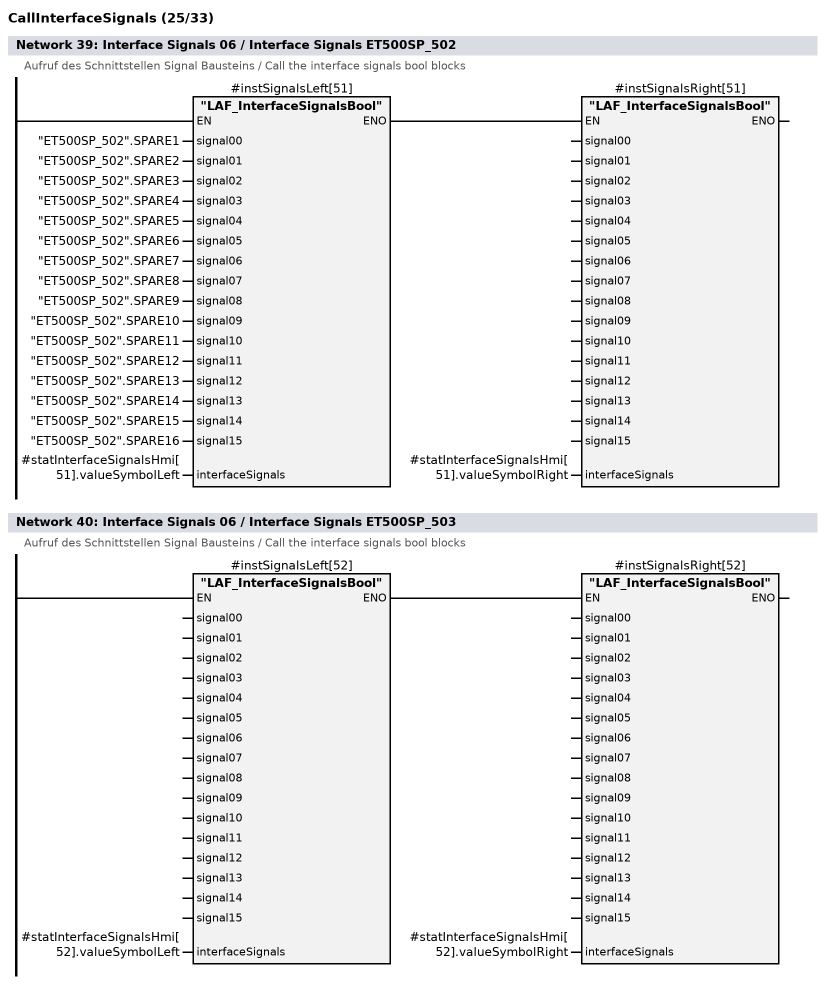
   RUNG wire#powerrail
      #instSignalsLeft[51](signal00 := "ET500SP_502".SPARE1, signal01 := "ET500SP_502".SPARE2, signal02 := "ET500SP_502".SPARE3, signal03 := "ET500SP_502".SPARE4, signal04 := "ET500SP_502".SPARE5, signal05 := "ET500SP_502".SPARE6, signal06 := "ET500SP_502".SPARE7, signal07 := "ET500SP_502".SPARE8, signal08 := "ET500SP_502".SPARE9, signal09 := "ET500SP_502".SPARE10, signal10 := "ET500SP_502".SPARE11, signal11 := "ET500SP_502".SPARE12, signal12 := "ET500SP_502".SPARE13, signal13 := "ET500SP_502".SPARE14, signal14 := "ET500SP_502".SPARE15, signal15 := "ET500SP_502".SPARE16, interfaceSignals := #statInterfaceSignalsHmi[51].valueSymbolLeft)
      #instSignalsRight[51](signal00 :=, signal01 :=, signal02 :=, signal03 :=, signal04 :=, signal05 :=, signal06 :=, signal07 :=, signal08 :=, signal09 :=, signal10 :=, signal11 :=, signal12 :=, signal13 :=, signal14 :=, signal15 :=, interfaceSignals := #statInterfaceSignalsHmi[51].valueSymbolRight)
   END_RUNG
   // the same network as SCL:
   #instSignalsLeft[51](signal00 := "ET500SP_502".SPARE1,   // "LAF_InterfaceSignalsBool"
                        signal01 := "ET500SP_502".SPARE2,
                        signal02 := "ET500SP_502".SPARE3,
                        signal03 := "ET500SP_502".SPARE4,
                        signal04 := "ET500SP_502".SPARE5,
                        signal05 := "ET500SP_502".SPARE6,
                        signal06 := "ET500SP_502".SPARE7,
                        signal07 := "ET500SP_502".SPARE8,
                        signal08 := "ET500SP_502".SPARE9,
                        signal09 := "ET500SP_502".SPARE10,
                        signal10 := "ET500SP_502".SPARE11,
                        signal11 := "ET500SP_502".SPARE12,
                        signal12 := "ET500SP_502".SPARE13,
                        signal13 := "ET500SP_502".SPARE14,
                        signal14 := "ET500SP_502".SPARE15,
                        signal15 := "ET500SP_502".SPARE16,
                        interfaceSignals := #statInterfaceSignalsHmi[51].valueSymbolLeft,
                        ENO => #_w1);
   IF #_w1 THEN
       #instSignalsRight[51](interfaceSignals := #statInterfaceSignalsHmi[51].valueSymbolRight);   // "LAF_InterfaceSignalsBool"
   END_IF;
END_REGION

REGION Network 40: Interface Signals 06 / Interface Signals ET500SP_503
   // Aufruf des Schnittstellen Signal Bausteins / Call the interface signals bool blocks
   RUNG wire#powerrail
      #instSignalsLeft[52](signal00 :=, signal01 :=, signal02 :=, signal03 :=, signal04 :=, signal05 :=, signal06 :=, signal07 :=, signal08 :=, signal09 :=, signal10 :=, signal11 :=, signal12 :=, signal13 :=, signal14 :=, signal15 :=, interfaceSignals := #statInterfaceSignalsHmi[52].valueSymbolLeft)
      #instSignalsRight[52](signal00 :=, signal01 :=, signal02 :=, signal03 :=, signal04 :=, signal05 :=, signal06 :=, signal07 :=, signal08 :=, signal09 :=, signal10 :=, signal11 :=, signal12 :=, signal13 :=, signal14 :=, signal15 :=, interfaceSignals := #statInterfaceSignalsHmi[52].valueSymbolRight)
   END_RUNG
   // the same network as SCL:
   #instSignalsLeft[52](interfaceSignals := #statInterfaceSignalsHmi[52].valueSymbolLeft, ENO => #_w1);   // "LAF_InterfaceSignalsBool"
   IF #_w1 THEN
       #instSignalsRight[52](interfaceSignals := #statInterfaceSignalsHmi[52].valueSymbolRight);   // "LAF_InterfaceSignalsBool"
   END_IF;
END_REGION

REGION Network 41: Interface Signals 06 / Interface Signals ET500SP_504
   // Aufruf des Schnittstellen Signal Bausteins / Call the interface signals bool blocks
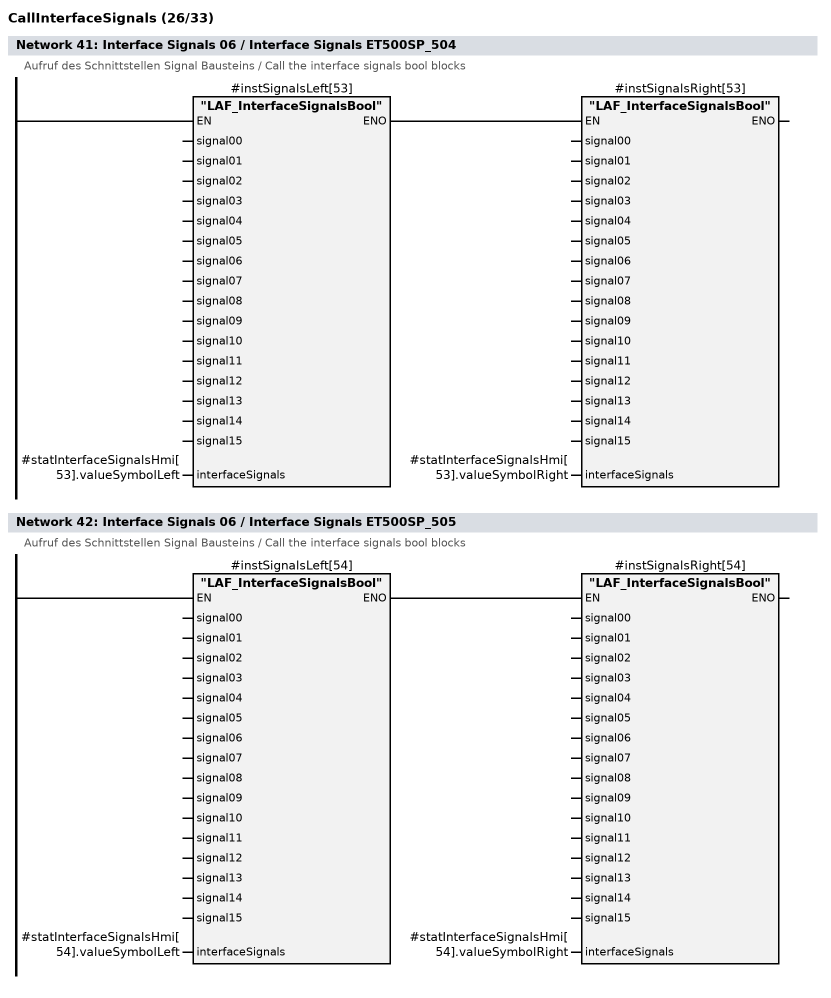
   RUNG wire#powerrail
      #instSignalsLeft[53](signal00 :=, signal01 :=, signal02 :=, signal03 :=, signal04 :=, signal05 :=, signal06 :=, signal07 :=, signal08 :=, signal09 :=, signal10 :=, signal11 :=, signal12 :=, signal13 :=, signal14 :=, signal15 :=, interfaceSignals := #statInterfaceSignalsHmi[53].valueSymbolLeft)
      #instSignalsRight[53](signal00 :=, signal01 :=, signal02 :=, signal03 :=, signal04 :=, signal05 :=, signal06 :=, signal07 :=, signal08 :=, signal09 :=, signal10 :=, signal11 :=, signal12 :=, signal13 :=, signal14 :=, signal15 :=, interfaceSignals := #statInterfaceSignalsHmi[53].valueSymbolRight)
   END_RUNG
   // the same network as SCL:
   #instSignalsLeft[53](interfaceSignals := #statInterfaceSignalsHmi[53].valueSymbolLeft, ENO => #_w1);   // "LAF_InterfaceSignalsBool"
   IF #_w1 THEN
       #instSignalsRight[53](interfaceSignals := #statInterfaceSignalsHmi[53].valueSymbolRight);   // "LAF_InterfaceSignalsBool"
   END_IF;
END_REGION

REGION Network 42: Interface Signals 06 / Interface Signals ET500SP_505
   // Aufruf des Schnittstellen Signal Bausteins / Call the interface signals bool blocks
   RUNG wire#powerrail
      #instSignalsLeft[54](signal00 :=, signal01 :=, signal02 :=, signal03 :=, signal04 :=, signal05 :=, signal06 :=, signal07 :=, signal08 :=, signal09 :=, signal10 :=, signal11 :=, signal12 :=, signal13 :=, signal14 :=, signal15 :=, interfaceSignals := #statInterfaceSignalsHmi[54].valueSymbolLeft)
      #instSignalsRight[54](signal00 :=, signal01 :=, signal02 :=, signal03 :=, signal04 :=, signal05 :=, signal06 :=, signal07 :=, signal08 :=, signal09 :=, signal10 :=, signal11 :=, signal12 :=, signal13 :=, signal14 :=, signal15 :=, interfaceSignals := #statInterfaceSignalsHmi[54].valueSymbolRight)
   END_RUNG
   // the same network as SCL:
   #instSignalsLeft[54](interfaceSignals := #statInterfaceSignalsHmi[54].valueSymbolLeft, ENO => #_w1);   // "LAF_InterfaceSignalsBool"
   IF #_w1 THEN
       #instSignalsRight[54](interfaceSignals := #statInterfaceSignalsHmi[54].valueSymbolRight);   // "LAF_InterfaceSignalsBool"
   END_IF;
END_REGION

REGION Network 43: Interface Signals 06 / Interface Signals ET500SP_506
   // Aufruf des Schnittstellen Signal Bausteins / Call the interface signals bool blocks
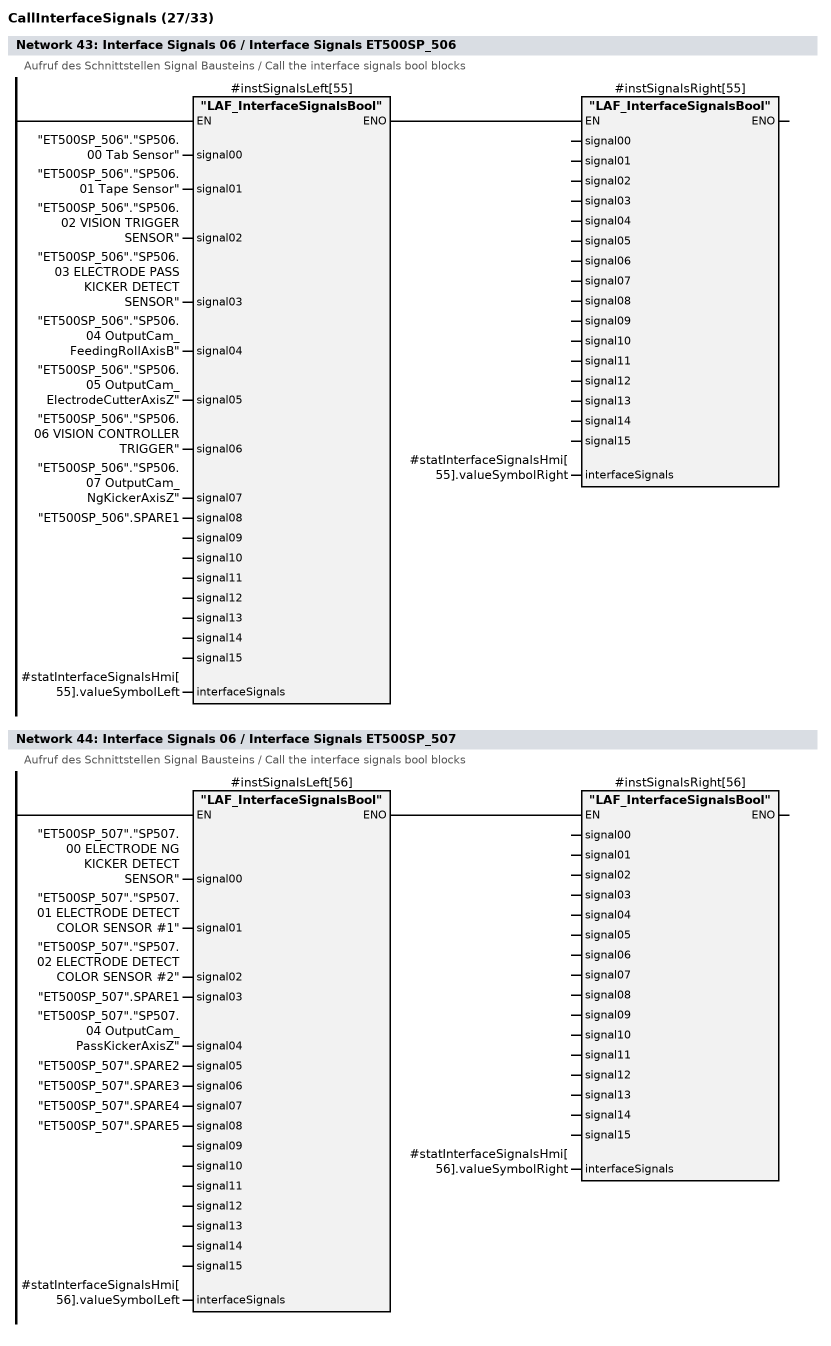
   RUNG wire#powerrail
      #instSignalsLeft[55](signal00 := "ET500SP_506"."SP506.00 Tab Sensor", signal01 := "ET500SP_506"."SP506.01 Tape Sensor", signal02 := "ET500SP_506"."SP506.02 VISION TRIGGER SENSOR", signal03 := "ET500SP_506"."SP506.03 ELECTRODE PASS KICKER DETECT SENSOR", signal04 := "ET500SP_506"."SP506.04 OutputCam_FeedingRollAxisB", signal05 := "ET500SP_506"."SP506.05 OutputCam_ElectrodeCutterAxisZ", signal06 := "ET500SP_506"."SP506.06 VISION CONTROLLER TRIGGER", signal07 := "ET500SP_506"."SP506.07 OutputCam_NgKickerAxisZ", signal08 := "ET500SP_506".SPARE1, signal09 :=, signal10 :=, signal11 :=, signal12 :=, signal13 :=, signal14 :=, signal15 :=, interfaceSignals := #statInterfaceSignalsHmi[55].valueSymbolLeft)
      #instSignalsRight[55](signal00 :=, signal01 :=, signal02 :=, signal03 :=, signal04 :=, signal05 :=, signal06 :=, signal07 :=, signal08 :=, signal09 :=, signal10 :=, signal11 :=, signal12 :=, signal13 :=, signal14 :=, signal15 :=, interfaceSignals := #statInterfaceSignalsHmi[55].valueSymbolRight)
   END_RUNG
   // the same network as SCL:
   #instSignalsLeft[55](signal00 := "ET500SP_506"."SP506.00 Tab Sensor",   // "LAF_InterfaceSignalsBool"
                        signal01 := "ET500SP_506"."SP506.01 Tape Sensor",
                        signal02 := "ET500SP_506"."SP506.02 VISION TRIGGER SENSOR",
                        signal03 := "ET500SP_506"."SP506.03 ELECTRODE PASS KICKER DETECT SENSOR",
                        signal04 := "ET500SP_506"."SP506.04 OutputCam_FeedingRollAxisB",
                        signal05 := "ET500SP_506"."SP506.05 OutputCam_ElectrodeCutterAxisZ",
                        signal06 := "ET500SP_506"."SP506.06 VISION CONTROLLER TRIGGER",
                        signal07 := "ET500SP_506"."SP506.07 OutputCam_NgKickerAxisZ",
                        signal08 := "ET500SP_506".SPARE1,
                        interfaceSignals := #statInterfaceSignalsHmi[55].valueSymbolLeft,
                        ENO => #_w1);
   IF #_w1 THEN
       #instSignalsRight[55](interfaceSignals := #statInterfaceSignalsHmi[55].valueSymbolRight);   // "LAF_InterfaceSignalsBool"
   END_IF;
END_REGION

REGION Network 44: Interface Signals 06 / Interface Signals ET500SP_507
   // Aufruf des Schnittstellen Signal Bausteins / Call the interface signals bool blocks
   RUNG wire#powerrail
      #instSignalsLeft[56](signal00 := "ET500SP_507"."SP507.00 ELECTRODE NG KICKER DETECT SENSOR", signal01 := "ET500SP_507"."SP507.01 ELECTRODE DETECT COLOR SENSOR #1", signal02 := "ET500SP_507"."SP507.02 ELECTRODE DETECT COLOR SENSOR #2", signal03 := "ET500SP_507".SPARE1, signal04 := "ET500SP_507"."SP507.04 OutputCam_PassKickerAxisZ", signal05 := "ET500SP_507".SPARE2, signal06 := "ET500SP_507".SPARE3, signal07 := "ET500SP_507".SPARE4, signal08 := "ET500SP_507".SPARE5, signal09 :=, signal10 :=, signal11 :=, signal12 :=, signal13 :=, signal14 :=, signal15 :=, interfaceSignals := #statInterfaceSignalsHmi[56].valueSymbolLeft)
      #instSignalsRight[56](signal00 :=, signal01 :=, signal02 :=, signal03 :=, signal04 :=, signal05 :=, signal06 :=, signal07 :=, signal08 :=, signal09 :=, signal10 :=, signal11 :=, signal12 :=, signal13 :=, signal14 :=, signal15 :=, interfaceSignals := #statInterfaceSignalsHmi[56].valueSymbolRight)
   END_RUNG
   // the same network as SCL:
   #instSignalsLeft[56](signal00 := "ET500SP_507"."SP507.00 ELECTRODE NG KICKER DETECT SENSOR",   // "LAF_InterfaceSignalsBool"
                        signal01 := "ET500SP_507"."SP507.01 ELECTRODE DETECT COLOR SENSOR #1",
                        signal02 := "ET500SP_507"."SP507.02 ELECTRODE DETECT COLOR SENSOR #2",
                        signal03 := "ET500SP_507".SPARE1,
                        signal04 := "ET500SP_507"."SP507.04 OutputCam_PassKickerAxisZ",
                        signal05 := "ET500SP_507".SPARE2,
                        signal06 := "ET500SP_507".SPARE3,
                        signal07 := "ET500SP_507".SPARE4,
                        signal08 := "ET500SP_507".SPARE5,
                        interfaceSignals := #statInterfaceSignalsHmi[56].valueSymbolLeft,
                        ENO => #_w1);
   IF #_w1 THEN
       #instSignalsRight[56](interfaceSignals := #statInterfaceSignalsHmi[56].valueSymbolRight);   // "LAF_InterfaceSignalsBool"
   END_IF;
END_REGION

REGION Network 45: Interface Signals 06 / Interface Signals ET500SP_508
   // Aufruf des Schnittstellen Signal Bausteins / Call the interface signals bool blocks
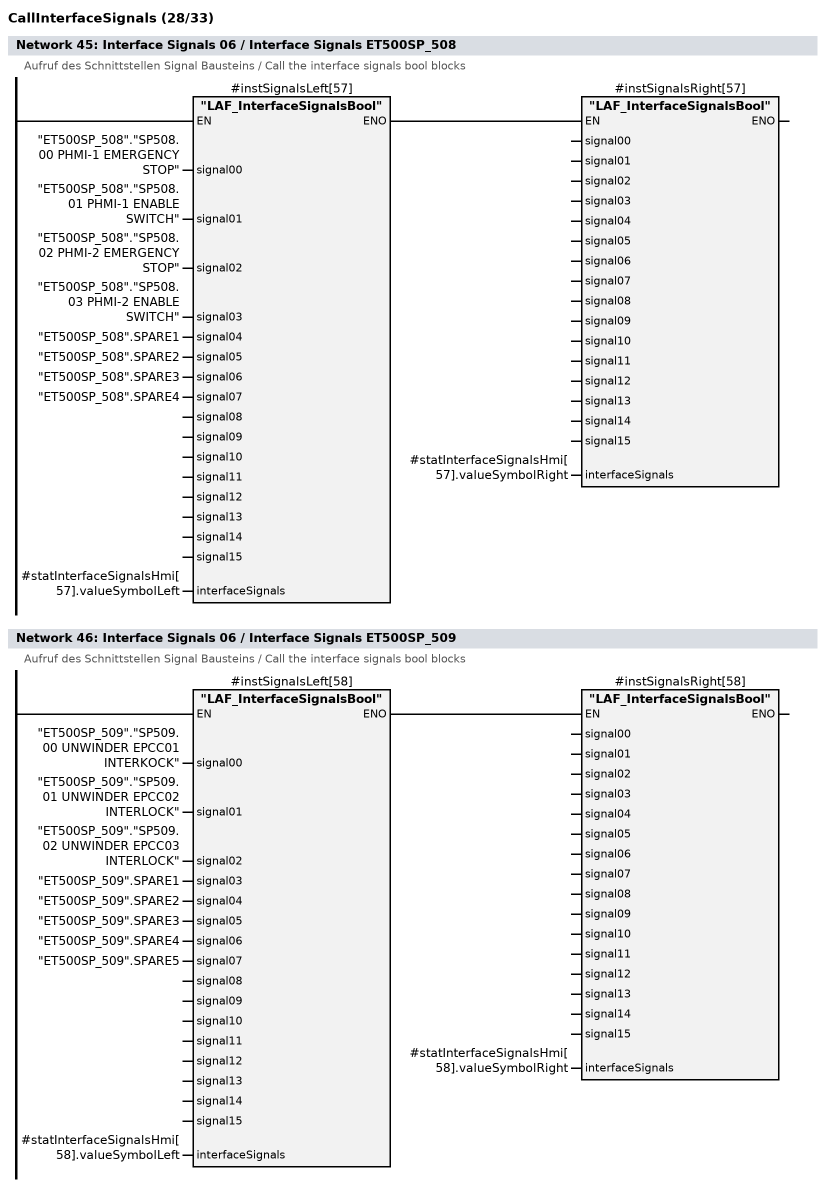
   RUNG wire#powerrail
      #instSignalsLeft[57](signal00 := "ET500SP_508"."SP508.00 PHMI-1 EMERGENCY STOP", signal01 := "ET500SP_508"."SP508.01 PHMI-1 ENABLE SWITCH", signal02 := "ET500SP_508"."SP508.02 PHMI-2 EMERGENCY STOP", signal03 := "ET500SP_508"."SP508.03 PHMI-2 ENABLE SWITCH", signal04 := "ET500SP_508".SPARE1, signal05 := "ET500SP_508".SPARE2, signal06 := "ET500SP_508".SPARE3, signal07 := "ET500SP_508".SPARE4, signal08 :=, signal09 :=, signal10 :=, signal11 :=, signal12 :=, signal13 :=, signal14 :=, signal15 :=, interfaceSignals := #statInterfaceSignalsHmi[57].valueSymbolLeft)
      #instSignalsRight[57](signal00 :=, signal01 :=, signal02 :=, signal03 :=, signal04 :=, signal05 :=, signal06 :=, signal07 :=, signal08 :=, signal09 :=, signal10 :=, signal11 :=, signal12 :=, signal13 :=, signal14 :=, signal15 :=, interfaceSignals := #statInterfaceSignalsHmi[57].valueSymbolRight)
   END_RUNG
   // the same network as SCL:
   #instSignalsLeft[57](signal00 := "ET500SP_508"."SP508.00 PHMI-1 EMERGENCY STOP",   // "LAF_InterfaceSignalsBool"
                        signal01 := "ET500SP_508"."SP508.01 PHMI-1 ENABLE SWITCH",
                        signal02 := "ET500SP_508"."SP508.02 PHMI-2 EMERGENCY STOP",
                        signal03 := "ET500SP_508"."SP508.03 PHMI-2 ENABLE SWITCH",
                        signal04 := "ET500SP_508".SPARE1,
                        signal05 := "ET500SP_508".SPARE2,
                        signal06 := "ET500SP_508".SPARE3,
                        signal07 := "ET500SP_508".SPARE4,
                        interfaceSignals := #statInterfaceSignalsHmi[57].valueSymbolLeft,
                        ENO => #_w1);
   IF #_w1 THEN
       #instSignalsRight[57](interfaceSignals := #statInterfaceSignalsHmi[57].valueSymbolRight);   // "LAF_InterfaceSignalsBool"
   END_IF;
END_REGION

REGION Network 46: Interface Signals 06 / Interface Signals ET500SP_509
   // Aufruf des Schnittstellen Signal Bausteins / Call the interface signals bool blocks
   RUNG wire#powerrail
      #instSignalsLeft[58](signal00 := "ET500SP_509"."SP509.00 UNWINDER EPCC01 INTERKOCK", signal01 := "ET500SP_509"."SP509.01 UNWINDER EPCC02 INTERLOCK", signal02 := "ET500SP_509"."SP509.02 UNWINDER EPCC03 INTERLOCK", signal03 := "ET500SP_509".SPARE1, signal04 := "ET500SP_509".SPARE2, signal05 := "ET500SP_509".SPARE3, signal06 := "ET500SP_509".SPARE4, signal07 := "ET500SP_509".SPARE5, signal08 :=, signal09 :=, signal10 :=, signal11 :=, signal12 :=, signal13 :=, signal14 :=, signal15 :=, interfaceSignals := #statInterfaceSignalsHmi[58].valueSymbolLeft)
      #instSignalsRight[58](signal00 :=, signal01 :=, signal02 :=, signal03 :=, signal04 :=, signal05 :=, signal06 :=, signal07 :=, signal08 :=, signal09 :=, signal10 :=, signal11 :=, signal12 :=, signal13 :=, signal14 :=, signal15 :=, interfaceSignals := #statInterfaceSignalsHmi[58].valueSymbolRight)
   END_RUNG
   // the same network as SCL:
   #instSignalsLeft[58](signal00 := "ET500SP_509"."SP509.00 UNWINDER EPCC01 INTERKOCK",   // "LAF_InterfaceSignalsBool"
                        signal01 := "ET500SP_509"."SP509.01 UNWINDER EPCC02 INTERLOCK",
                        signal02 := "ET500SP_509"."SP509.02 UNWINDER EPCC03 INTERLOCK",
                        signal03 := "ET500SP_509".SPARE1,
                        signal04 := "ET500SP_509".SPARE2,
                        signal05 := "ET500SP_509".SPARE3,
                        signal06 := "ET500SP_509".SPARE4,
                        signal07 := "ET500SP_509".SPARE5,
                        interfaceSignals := #statInterfaceSignalsHmi[58].valueSymbolLeft,
                        ENO => #_w1);
   IF #_w1 THEN
       #instSignalsRight[58](interfaceSignals := #statInterfaceSignalsHmi[58].valueSymbolRight);   // "LAF_InterfaceSignalsBool"
   END_IF;
END_REGION

REGION Network 47: Interface Signals 06 / Interface Signals ET500SP_513
   // Aufruf des Schnittstellen Signal Bausteins / Call the interface signals bool blocks
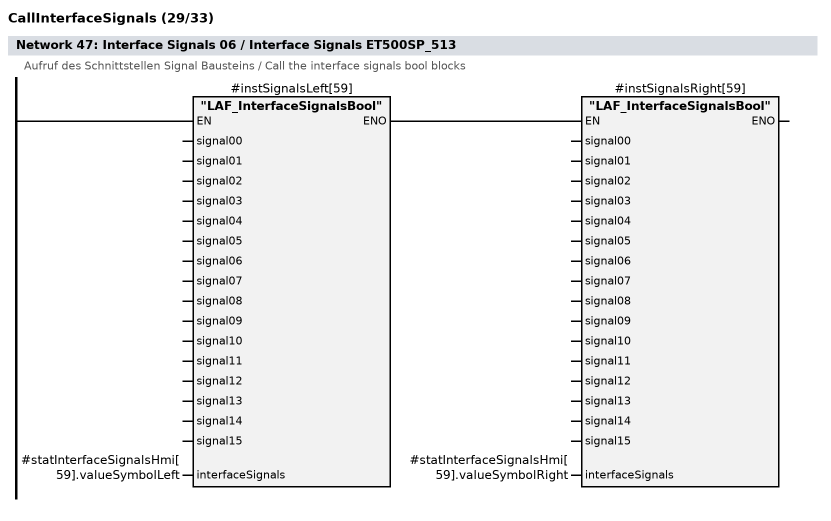
   RUNG wire#powerrail
      #instSignalsLeft[59](signal00 :=, signal01 :=, signal02 :=, signal03 :=, signal04 :=, signal05 :=, signal06 :=, signal07 :=, signal08 :=, signal09 :=, signal10 :=, signal11 :=, signal12 :=, signal13 :=, signal14 :=, signal15 :=, interfaceSignals := #statInterfaceSignalsHmi[59].valueSymbolLeft)
      #instSignalsRight[59](signal00 :=, signal01 :=, signal02 :=, signal03 :=, signal04 :=, signal05 :=, signal06 :=, signal07 :=, signal08 :=, signal09 :=, signal10 :=, signal11 :=, signal12 :=, signal13 :=, signal14 :=, signal15 :=, interfaceSignals := #statInterfaceSignalsHmi[59].valueSymbolRight)
   END_RUNG
   // the same network as SCL:
   #instSignalsLeft[59](interfaceSignals := #statInterfaceSignalsHmi[59].valueSymbolLeft, ENO => #_w1);   // "LAF_InterfaceSignalsBool"
   IF #_w1 THEN
       #instSignalsRight[59](interfaceSignals := #statInterfaceSignalsHmi[59].valueSymbolRight);   // "LAF_InterfaceSignalsBool"
   END_IF;
END_REGION

REGION Network 48: Interface Signals 06 / Interface Signals CPU DI1
   // Aufruf des Schnittstellen Signal Bausteins / Call the interface signals bool blocks
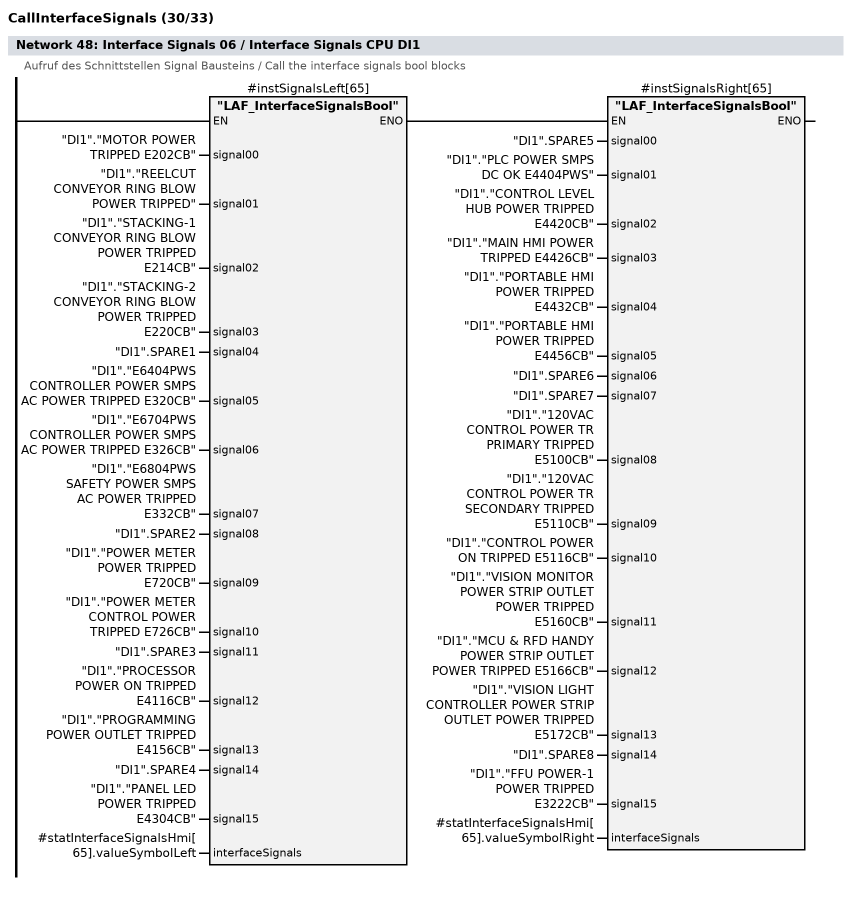
   RUNG wire#powerrail
      #instSignalsLeft[65](signal00 := "DI1"."MOTOR POWER TRIPPED E202CB", signal01 := "DI1"."REELCUT CONVEYOR RING BLOW POWER TRIPPED", signal02 := "DI1"."STACKING-1 CONVEYOR RING BLOW POWER TRIPPED E214CB", signal03 := "DI1"."STACKING-2 CONVEYOR RING BLOW POWER TRIPPED E220CB", signal04 := "DI1".SPARE1, signal05 := "DI1"."E6404PWS CONTROLLER POWER SMPS AC POWER TRIPPED E320CB", signal06 := "DI1"."E6704PWS CONTROLLER POWER SMPS AC POWER TRIPPED E326CB", signal07 := "DI1"."E6804PWS SAFETY POWER SMPS AC POWER TRIPPED E332CB", signal08 := "DI1".SPARE2, signal09 := "DI1"."POWER METER POWER TRIPPED E720CB", signal10 := "DI1"."POWER METER CONTROL POWER TRIPPED E726CB", signal11 := "DI1".SPARE3, signal12 := "DI1"."PROCESSOR POWER ON TRIPPED E4116CB", signal13 := "DI1"."PROGRAMMING POWER OUTLET TRIPPED E4156CB", signal14 := "DI1".SPARE4, signal15 := "DI1"."PANEL LED POWER TRIPPED E4304CB", interfaceSignals := #statInterfaceSignalsHmi[65].valueSymbolLeft)
      #instSignalsRight[65](signal00 := "DI1".SPARE5, signal01 := "DI1"."PLC POWER SMPS DC OK E4404PWS", signal02 := "DI1"."CONTROL LEVEL HUB POWER TRIPPED E4420CB", signal03 := "DI1"."MAIN HMI POWER TRIPPED E4426CB", signal04 := "DI1"."PORTABLE HMI POWER TRIPPED E4432CB", signal05 := "DI1"."PORTABLE HMI POWER TRIPPED E4456CB", signal06 := "DI1".SPARE6, signal07 := "DI1".SPARE7, signal08 := "DI1"."120VAC CONTROL POWER TR PRIMARY TRIPPED E5100CB", signal09 := "DI1"."120VAC CONTROL POWER TR SECONDARY TRIPPED E5110CB", signal10 := "DI1"."CONTROL POWER ON TRIPPED E5116CB", signal11 := "DI1"."VISION MONITOR POWER STRIP OUTLET POWER TRIPPED E5160CB", signal12 := "DI1"."MCU & RFD HANDY POWER STRIP OUTLET POWER TRIPPED E5166CB", signal13 := "DI1"."VISION LIGHT CONTROLLER POWER STRIP OUTLET POWER TRIPPED E5172CB", signal14 := "DI1".SPARE8, signal15 := "DI1"."FFU POWER-1 POWER TRIPPED E3222CB", interfaceSignals := #statInterfaceSignalsHmi[65].valueSymbolRight)
   END_RUNG
   // the same network as SCL:
   #instSignalsLeft[65](signal00 := "DI1"."MOTOR POWER TRIPPED E202CB",   // "LAF_InterfaceSignalsBool"
                        signal01 := "DI1"."REELCUT CONVEYOR RING BLOW POWER TRIPPED",
                        signal02 := "DI1"."STACKING-1 CONVEYOR RING BLOW POWER TRIPPED E214CB",
                        signal03 := "DI1"."STACKING-2 CONVEYOR RING BLOW POWER TRIPPED E220CB",
                        signal04 := "DI1".SPARE1,
                        signal05 := "DI1"."E6404PWS CONTROLLER POWER SMPS AC POWER TRIPPED E320CB",
                        signal06 := "DI1"."E6704PWS CONTROLLER POWER SMPS AC POWER TRIPPED E326CB",
                        signal07 := "DI1"."E6804PWS SAFETY POWER SMPS AC POWER TRIPPED E332CB",
                        signal08 := "DI1".SPARE2,
                        signal09 := "DI1"."POWER METER POWER TRIPPED E720CB",
                        signal10 := "DI1"."POWER METER CONTROL POWER TRIPPED E726CB",
                        signal11 := "DI1".SPARE3,
                        signal12 := "DI1"."PROCESSOR POWER ON TRIPPED E4116CB",
                        signal13 := "DI1"."PROGRAMMING POWER OUTLET TRIPPED E4156CB",
                        signal14 := "DI1".SPARE4,
                        signal15 := "DI1"."PANEL LED POWER TRIPPED E4304CB",
                        interfaceSignals := #statInterfaceSignalsHmi[65].valueSymbolLeft,
                        ENO => #_w1);
   IF #_w1 THEN
       #instSignalsRight[65](signal00 := "DI1".SPARE5,   // "LAF_InterfaceSignalsBool"
                             signal01 := "DI1"."PLC POWER SMPS DC OK E4404PWS",
                             signal02 := "DI1"."CONTROL LEVEL HUB POWER TRIPPED E4420CB",
                             signal03 := "DI1"."MAIN HMI POWER TRIPPED E4426CB",
                             signal04 := "DI1"."PORTABLE HMI POWER TRIPPED E4432CB",
                             signal05 := "DI1"."PORTABLE HMI POWER TRIPPED E4456CB",
                             signal06 := "DI1".SPARE6,
                             signal07 := "DI1".SPARE7,
                             signal08 := "DI1"."120VAC CONTROL POWER TR PRIMARY TRIPPED E5100CB",
                             signal09 := "DI1"."120VAC CONTROL POWER TR SECONDARY TRIPPED E5110CB",
                             signal10 := "DI1"."CONTROL POWER ON TRIPPED E5116CB",
                             signal11 := "DI1"."VISION MONITOR POWER STRIP OUTLET POWER TRIPPED E5160CB",
                             signal12 := "DI1"."MCU & RFD HANDY POWER STRIP OUTLET POWER TRIPPED E5166CB",
                             signal13 := "DI1"."VISION LIGHT CONTROLLER POWER STRIP OUTLET POWER TRIPPED E5172CB",
                             signal14 := "DI1".SPARE8,
                             signal15 := "DI1"."FFU POWER-1 POWER TRIPPED E3222CB",
                             interfaceSignals := #statInterfaceSignalsHmi[65].valueSymbolRight);
   END_IF;
END_REGION

REGION Network 49: Interface Signals 06 / Interface Signals CPU DI2
   // Aufruf des Schnittstellen Signal Bausteins / Call the interface signals bool blocks
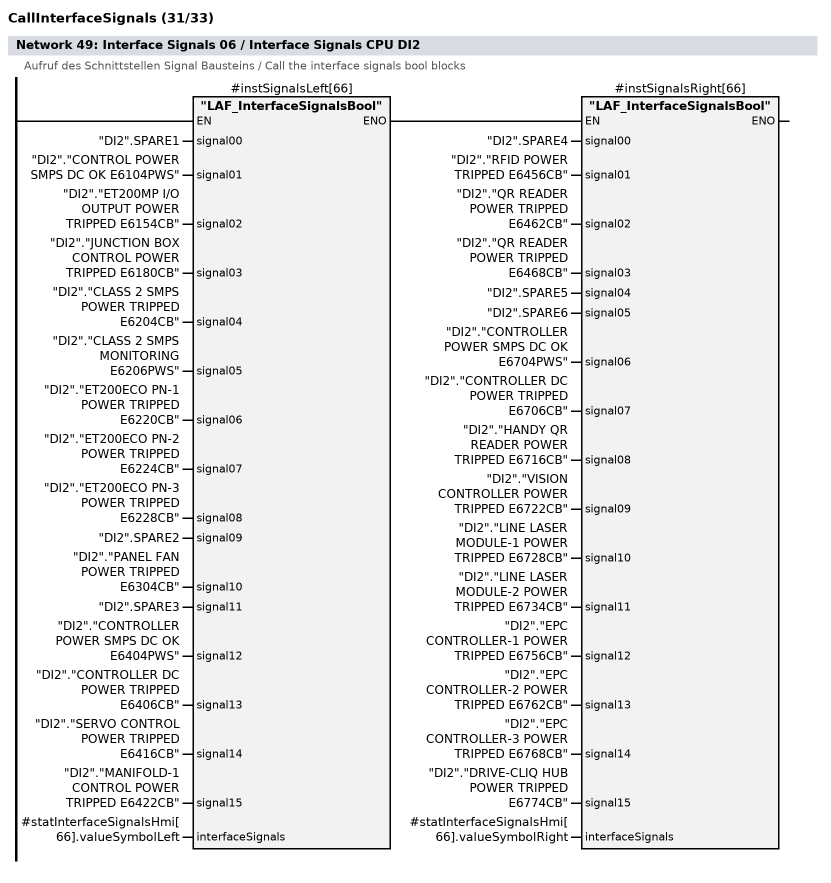
   RUNG wire#powerrail
      #instSignalsLeft[66](signal00 := "DI2".SPARE1, signal01 := "DI2"."CONTROL POWER SMPS DC OK E6104PWS", signal02 := "DI2"."ET200MP I/O OUTPUT POWER TRIPPED E6154CB", signal03 := "DI2"."JUNCTION BOX CONTROL POWER TRIPPED E6180CB", signal04 := "DI2"."CLASS 2 SMPS POWER TRIPPED E6204CB", signal05 := "DI2"."CLASS 2 SMPS MONITORING E6206PWS", signal06 := "DI2"."ET200ECO PN-1 POWER TRIPPED E6220CB", signal07 := "DI2"."ET200ECO PN-2 POWER TRIPPED E6224CB", signal08 := "DI2"."ET200ECO PN-3 POWER TRIPPED E6228CB", signal09 := "DI2".SPARE2, signal10 := "DI2"."PANEL FAN POWER TRIPPED E6304CB", signal11 := "DI2".SPARE3, signal12 := "DI2"."CONTROLLER POWER SMPS DC OK E6404PWS", signal13 := "DI2"."CONTROLLER DC POWER TRIPPED E6406CB", signal14 := "DI2"."SERVO CONTROL POWER TRIPPED E6416CB", signal15 := "DI2"."MANIFOLD-1 CONTROL POWER TRIPPED E6422CB", interfaceSignals := #statInterfaceSignalsHmi[66].valueSymbolLeft)
      #instSignalsRight[66](signal00 := "DI2".SPARE4, signal01 := "DI2"."RFID POWER TRIPPED E6456CB", signal02 := "DI2"."QR READER POWER TRIPPED E6462CB", signal03 := "DI2"."QR READER POWER TRIPPED E6468CB", signal04 := "DI2".SPARE5, signal05 := "DI2".SPARE6, signal06 := "DI2"."CONTROLLER POWER SMPS DC OK E6704PWS", signal07 := "DI2"."CONTROLLER DC POWER TRIPPED E6706CB", signal08 := "DI2"."HANDY QR READER POWER TRIPPED E6716CB", signal09 := "DI2"."VISION CONTROLLER POWER TRIPPED E6722CB", signal10 := "DI2"."LINE LASER MODULE-1 POWER TRIPPED E6728CB", signal11 := "DI2"."LINE LASER MODULE-2 POWER TRIPPED E6734CB", signal12 := "DI2"."EPC CONTROLLER-1 POWER TRIPPED E6756CB", signal13 := "DI2"."EPC CONTROLLER-2 POWER TRIPPED E6762CB", signal14 := "DI2"."EPC CONTROLLER-3 POWER TRIPPED E6768CB", signal15 := "DI2"."DRIVE-CLIQ HUB POWER TRIPPED E6774CB", interfaceSignals := #statInterfaceSignalsHmi[66].valueSymbolRight)
   END_RUNG
   // the same network as SCL:
   #instSignalsLeft[66](signal00 := "DI2".SPARE1,   // "LAF_InterfaceSignalsBool"
                        signal01 := "DI2"."CONTROL POWER SMPS DC OK E6104PWS",
                        signal02 := "DI2"."ET200MP I/O OUTPUT POWER TRIPPED E6154CB",
                        signal03 := "DI2"."JUNCTION BOX CONTROL POWER TRIPPED E6180CB",
                        signal04 := "DI2"."CLASS 2 SMPS POWER TRIPPED E6204CB",
                        signal05 := "DI2"."CLASS 2 SMPS MONITORING E6206PWS",
                        signal06 := "DI2"."ET200ECO PN-1 POWER TRIPPED E6220CB",
                        signal07 := "DI2"."ET200ECO PN-2 POWER TRIPPED E6224CB",
                        signal08 := "DI2"."ET200ECO PN-3 POWER TRIPPED E6228CB",
                        signal09 := "DI2".SPARE2,
                        signal10 := "DI2"."PANEL FAN POWER TRIPPED E6304CB",
                        signal11 := "DI2".SPARE3,
                        signal12 := "DI2"."CONTROLLER POWER SMPS DC OK E6404PWS",
                        signal13 := "DI2"."CONTROLLER DC POWER TRIPPED E6406CB",
                        signal14 := "DI2"."SERVO CONTROL POWER TRIPPED E6416CB",
                        signal15 := "DI2"."MANIFOLD-1 CONTROL POWER TRIPPED E6422CB",
                        interfaceSignals := #statInterfaceSignalsHmi[66].valueSymbolLeft,
                        ENO => #_w1);
   IF #_w1 THEN
       #instSignalsRight[66](signal00 := "DI2".SPARE4,   // "LAF_InterfaceSignalsBool"
                             signal01 := "DI2"."RFID POWER TRIPPED E6456CB",
                             signal02 := "DI2"."QR READER POWER TRIPPED E6462CB",
                             signal03 := "DI2"."QR READER POWER TRIPPED E6468CB",
                             signal04 := "DI2".SPARE5,
                             signal05 := "DI2".SPARE6,
                             signal06 := "DI2"."CONTROLLER POWER SMPS DC OK E6704PWS",
                             signal07 := "DI2"."CONTROLLER DC POWER TRIPPED E6706CB",
                             signal08 := "DI2"."HANDY QR READER POWER TRIPPED E6716CB",
                             signal09 := "DI2"."VISION CONTROLLER POWER TRIPPED E6722CB",
                             signal10 := "DI2"."LINE LASER MODULE-1 POWER TRIPPED E6728CB",
                             signal11 := "DI2"."LINE LASER MODULE-2 POWER TRIPPED E6734CB",
                             signal12 := "DI2"."EPC CONTROLLER-1 POWER TRIPPED E6756CB",
                             signal13 := "DI2"."EPC CONTROLLER-2 POWER TRIPPED E6762CB",
                             signal14 := "DI2"."EPC CONTROLLER-3 POWER TRIPPED E6768CB",
                             signal15 := "DI2"."DRIVE-CLIQ HUB POWER TRIPPED E6774CB",
                             interfaceSignals := #statInterfaceSignalsHmi[66].valueSymbolRight);
   END_IF;
END_REGION

REGION Network 50: Interface Signals 06 / Interface Signals CPU DI3
   // Aufruf des Schnittstellen Signal Bausteins / Call the interface signals bool blocks
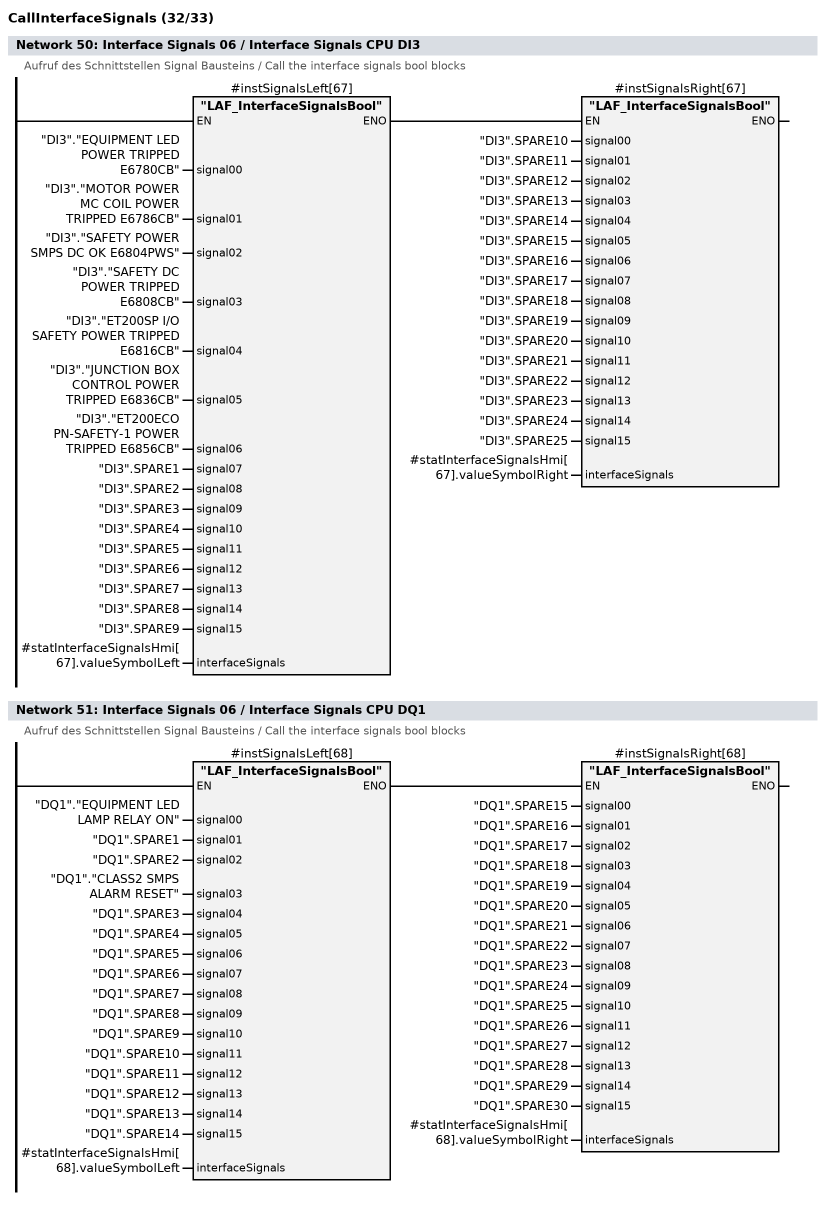
   RUNG wire#powerrail
      #instSignalsLeft[67](signal00 := "DI3"."EQUIPMENT LED POWER TRIPPED E6780CB", signal01 := "DI3"."MOTOR POWER MC COIL POWER TRIPPED E6786CB", signal02 := "DI3"."SAFETY POWER SMPS DC OK E6804PWS", signal03 := "DI3"."SAFETY DC POWER TRIPPED E6808CB", signal04 := "DI3"."ET200SP I/O SAFETY POWER TRIPPED E6816CB", signal05 := "DI3"."JUNCTION BOX CONTROL POWER TRIPPED E6836CB", signal06 := "DI3"."ET200ECO PN-SAFETY-1 POWER TRIPPED E6856CB", signal07 := "DI3".SPARE1, signal08 := "DI3".SPARE2, signal09 := "DI3".SPARE3, signal10 := "DI3".SPARE4, signal11 := "DI3".SPARE5, signal12 := "DI3".SPARE6, signal13 := "DI3".SPARE7, signal14 := "DI3".SPARE8, signal15 := "DI3".SPARE9, interfaceSignals := #statInterfaceSignalsHmi[67].valueSymbolLeft)
      #instSignalsRight[67](signal00 := "DI3".SPARE10, signal01 := "DI3".SPARE11, signal02 := "DI3".SPARE12, signal03 := "DI3".SPARE13, signal04 := "DI3".SPARE14, signal05 := "DI3".SPARE15, signal06 := "DI3".SPARE16, signal07 := "DI3".SPARE17, signal08 := "DI3".SPARE18, signal09 := "DI3".SPARE19, signal10 := "DI3".SPARE20, signal11 := "DI3".SPARE21, signal12 := "DI3".SPARE22, signal13 := "DI3".SPARE23, signal14 := "DI3".SPARE24, signal15 := "DI3".SPARE25, interfaceSignals := #statInterfaceSignalsHmi[67].valueSymbolRight)
   END_RUNG
   // the same network as SCL:
   #instSignalsLeft[67](signal00 := "DI3"."EQUIPMENT LED POWER TRIPPED E6780CB",   // "LAF_InterfaceSignalsBool"
                        signal01 := "DI3"."MOTOR POWER MC COIL POWER TRIPPED E6786CB",
                        signal02 := "DI3"."SAFETY POWER SMPS DC OK E6804PWS",
                        signal03 := "DI3"."SAFETY DC POWER TRIPPED E6808CB",
                        signal04 := "DI3"."ET200SP I/O SAFETY POWER TRIPPED E6816CB",
                        signal05 := "DI3"."JUNCTION BOX CONTROL POWER TRIPPED E6836CB",
                        signal06 := "DI3"."ET200ECO PN-SAFETY-1 POWER TRIPPED E6856CB",
                        signal07 := "DI3".SPARE1,
                        signal08 := "DI3".SPARE2,
                        signal09 := "DI3".SPARE3,
                        signal10 := "DI3".SPARE4,
                        signal11 := "DI3".SPARE5,
                        signal12 := "DI3".SPARE6,
                        signal13 := "DI3".SPARE7,
                        signal14 := "DI3".SPARE8,
                        signal15 := "DI3".SPARE9,
                        interfaceSignals := #statInterfaceSignalsHmi[67].valueSymbolLeft,
                        ENO => #_w1);
   IF #_w1 THEN
       #instSignalsRight[67](signal00 := "DI3".SPARE10,   // "LAF_InterfaceSignalsBool"
                             signal01 := "DI3".SPARE11,
                             signal02 := "DI3".SPARE12,
                             signal03 := "DI3".SPARE13,
                             signal04 := "DI3".SPARE14,
                             signal05 := "DI3".SPARE15,
                             signal06 := "DI3".SPARE16,
                             signal07 := "DI3".SPARE17,
                             signal08 := "DI3".SPARE18,
                             signal09 := "DI3".SPARE19,
                             signal10 := "DI3".SPARE20,
                             signal11 := "DI3".SPARE21,
                             signal12 := "DI3".SPARE22,
                             signal13 := "DI3".SPARE23,
                             signal14 := "DI3".SPARE24,
                             signal15 := "DI3".SPARE25,
                             interfaceSignals := #statInterfaceSignalsHmi[67].valueSymbolRight);
   END_IF;
END_REGION

REGION Network 51: Interface Signals 06 / Interface Signals CPU DQ1
   // Aufruf des Schnittstellen Signal Bausteins / Call the interface signals bool blocks
   RUNG wire#powerrail
      #instSignalsLeft[68](signal00 := "DQ1"."EQUIPMENT LED LAMP RELAY ON", signal01 := "DQ1".SPARE1, signal02 := "DQ1".SPARE2, signal03 := "DQ1"."CLASS2 SMPS ALARM RESET", signal04 := "DQ1".SPARE3, signal05 := "DQ1".SPARE4, signal06 := "DQ1".SPARE5, signal07 := "DQ1".SPARE6, signal08 := "DQ1".SPARE7, signal09 := "DQ1".SPARE8, signal10 := "DQ1".SPARE9, signal11 := "DQ1".SPARE10, signal12 := "DQ1".SPARE11, signal13 := "DQ1".SPARE12, signal14 := "DQ1".SPARE13, signal15 := "DQ1".SPARE14, interfaceSignals := #statInterfaceSignalsHmi[68].valueSymbolLeft)
      #instSignalsRight[68](signal00 := "DQ1".SPARE15, signal01 := "DQ1".SPARE16, signal02 := "DQ1".SPARE17, signal03 := "DQ1".SPARE18, signal04 := "DQ1".SPARE19, signal05 := "DQ1".SPARE20, signal06 := "DQ1".SPARE21, signal07 := "DQ1".SPARE22, signal08 := "DQ1".SPARE23, signal09 := "DQ1".SPARE24, signal10 := "DQ1".SPARE25, signal11 := "DQ1".SPARE26, signal12 := "DQ1".SPARE27, signal13 := "DQ1".SPARE28, signal14 := "DQ1".SPARE29, signal15 := "DQ1".SPARE30, interfaceSignals := #statInterfaceSignalsHmi[68].valueSymbolRight)
   END_RUNG
   // the same network as SCL:
   #instSignalsLeft[68](signal00 := "DQ1"."EQUIPMENT LED LAMP RELAY ON",   // "LAF_InterfaceSignalsBool"
                        signal01 := "DQ1".SPARE1,
                        signal02 := "DQ1".SPARE2,
                        signal03 := "DQ1"."CLASS2 SMPS ALARM RESET",
                        signal04 := "DQ1".SPARE3,
                        signal05 := "DQ1".SPARE4,
                        signal06 := "DQ1".SPARE5,
                        signal07 := "DQ1".SPARE6,
                        signal08 := "DQ1".SPARE7,
                        signal09 := "DQ1".SPARE8,
                        signal10 := "DQ1".SPARE9,
                        signal11 := "DQ1".SPARE10,
                        signal12 := "DQ1".SPARE11,
                        signal13 := "DQ1".SPARE12,
                        signal14 := "DQ1".SPARE13,
                        signal15 := "DQ1".SPARE14,
                        interfaceSignals := #statInterfaceSignalsHmi[68].valueSymbolLeft,
                        ENO => #_w1);
   IF #_w1 THEN
       #instSignalsRight[68](signal00 := "DQ1".SPARE15,   // "LAF_InterfaceSignalsBool"
                             signal01 := "DQ1".SPARE16,
                             signal02 := "DQ1".SPARE17,
                             signal03 := "DQ1".SPARE18,
                             signal04 := "DQ1".SPARE19,
                             signal05 := "DQ1".SPARE20,
                             signal06 := "DQ1".SPARE21,
                             signal07 := "DQ1".SPARE22,
                             signal08 := "DQ1".SPARE23,
                             signal09 := "DQ1".SPARE24,
                             signal10 := "DQ1".SPARE25,
                             signal11 := "DQ1".SPARE26,
                             signal12 := "DQ1".SPARE27,
                             signal13 := "DQ1".SPARE28,
                             signal14 := "DQ1".SPARE29,
                             signal15 := "DQ1".SPARE30,
                             interfaceSignals := #statInterfaceSignalsHmi[68].valueSymbolRight);
   END_IF;
END_REGION

REGION Network 52: Interface Signals 06 / Interface Signals CPU FDI1
   // Aufruf des Schnittstellen Signal Bausteins / Call the interface signals bool blocks
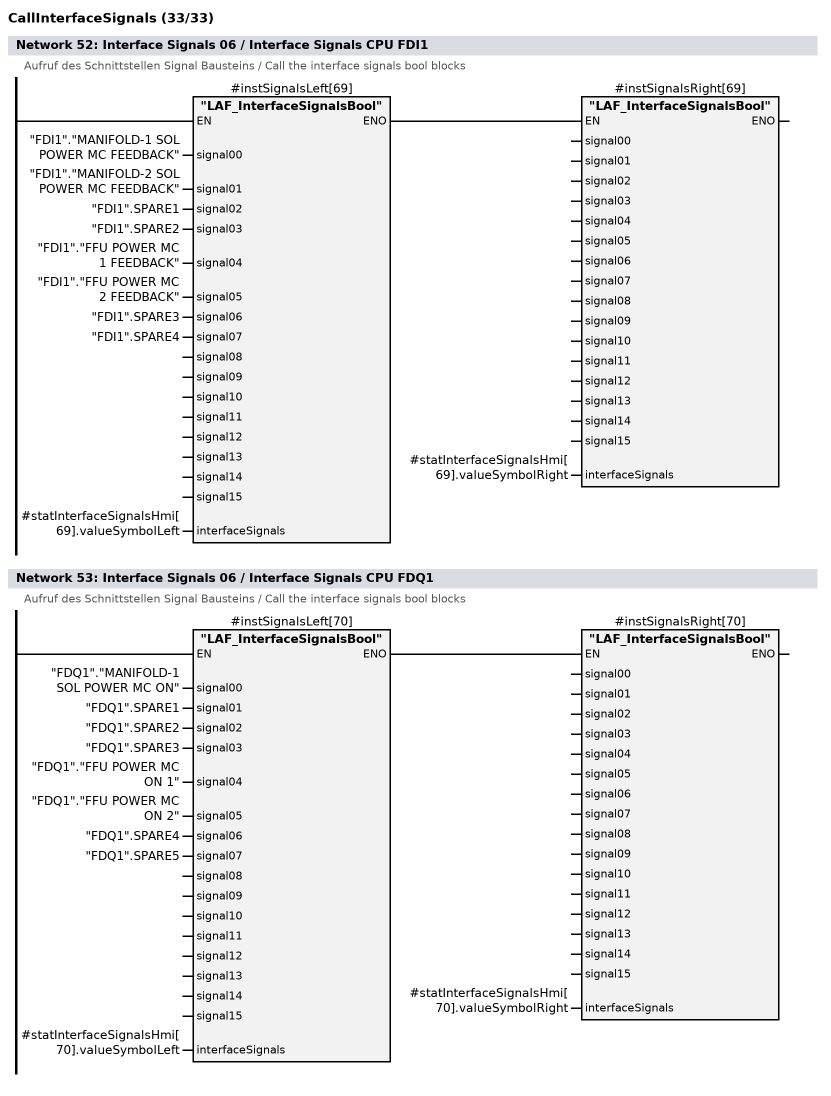
   RUNG wire#powerrail
      #instSignalsLeft[69](signal00 := "FDI1"."MANIFOLD-1 SOL POWER MC FEEDBACK", signal01 := "FDI1"."MANIFOLD-2 SOL POWER MC FEEDBACK", signal02 := "FDI1".SPARE1, signal03 := "FDI1".SPARE2, signal04 := "FDI1"."FFU POWER MC 1 FEEDBACK", signal05 := "FDI1"."FFU POWER MC 2 FEEDBACK", signal06 := "FDI1".SPARE3, signal07 := "FDI1".SPARE4, signal08 :=, signal09 :=, signal10 :=, signal11 :=, signal12 :=, signal13 :=, signal14 :=, signal15 :=, interfaceSignals := #statInterfaceSignalsHmi[69].valueSymbolLeft)
      #instSignalsRight[69](signal00 :=, signal01 :=, signal02 :=, signal03 :=, signal04 :=, signal05 :=, signal06 :=, signal07 :=, signal08 :=, signal09 :=, signal10 :=, signal11 :=, signal12 :=, signal13 :=, signal14 :=, signal15 :=, interfaceSignals := #statInterfaceSignalsHmi[69].valueSymbolRight)
   END_RUNG
   // the same network as SCL:
   #instSignalsLeft[69](signal00 := "FDI1"."MANIFOLD-1 SOL POWER MC FEEDBACK",   // "LAF_InterfaceSignalsBool"
                        signal01 := "FDI1"."MANIFOLD-2 SOL POWER MC FEEDBACK",
                        signal02 := "FDI1".SPARE1,
                        signal03 := "FDI1".SPARE2,
                        signal04 := "FDI1"."FFU POWER MC 1 FEEDBACK",
                        signal05 := "FDI1"."FFU POWER MC 2 FEEDBACK",
                        signal06 := "FDI1".SPARE3,
                        signal07 := "FDI1".SPARE4,
                        interfaceSignals := #statInterfaceSignalsHmi[69].valueSymbolLeft,
                        ENO => #_w1);
   IF #_w1 THEN
       #instSignalsRight[69](interfaceSignals := #statInterfaceSignalsHmi[69].valueSymbolRight);   // "LAF_InterfaceSignalsBool"
   END_IF;
END_REGION

REGION Network 53: Interface Signals 06 / Interface Signals CPU FDQ1
   // Aufruf des Schnittstellen Signal Bausteins / Call the interface signals bool blocks
   RUNG wire#powerrail
      #instSignalsLeft[70](signal00 := "FDQ1"."MANIFOLD-1 SOL POWER MC ON", signal01 := "FDQ1".SPARE1, signal02 := "FDQ1".SPARE2, signal03 := "FDQ1".SPARE3, signal04 := "FDQ1"."FFU POWER MC ON 1", signal05 := "FDQ1"."FFU POWER MC ON 2", signal06 := "FDQ1".SPARE4, signal07 := "FDQ1".SPARE5, signal08 :=, signal09 :=, signal10 :=, signal11 :=, signal12 :=, signal13 :=, signal14 :=, signal15 :=, interfaceSignals := #statInterfaceSignalsHmi[70].valueSymbolLeft)
      #instSignalsRight[70](signal00 :=, signal01 :=, signal02 :=, signal03 :=, signal04 :=, signal05 :=, signal06 :=, signal07 :=, signal08 :=, signal09 :=, signal10 :=, signal11 :=, signal12 :=, signal13 :=, signal14 :=, signal15 :=, interfaceSignals := #statInterfaceSignalsHmi[70].valueSymbolRight)
   END_RUNG
   // the same network as SCL:
   #instSignalsLeft[70](signal00 := "FDQ1"."MANIFOLD-1 SOL POWER MC ON",   // "LAF_InterfaceSignalsBool"
                        signal01 := "FDQ1".SPARE1,
                        signal02 := "FDQ1".SPARE2,
                        signal03 := "FDQ1".SPARE3,
                        signal04 := "FDQ1"."FFU POWER MC ON 1",
                        signal05 := "FDQ1"."FFU POWER MC ON 2",
                        signal06 := "FDQ1".SPARE4,
                        signal07 := "FDQ1".SPARE5,
                        interfaceSignals := #statInterfaceSignalsHmi[70].valueSymbolLeft,
                        ENO => #_w1);
   IF #_w1 THEN
       #instSignalsRight[70](interfaceSignals := #statInterfaceSignalsHmi[70].valueSymbolRight);   // "LAF_InterfaceSignalsBool"
   END_IF;
END_REGION
END_FUNCTION_BLOCK
